// TIA Portal V20 export
// export: Created 2025-12-01T14:57:27.0344131Z, ExportSetting None, DisplayName Totally Integrated Automation Portal, DisplayVersion V20 Update 3, DisplayName TIA Portal Openness, DisplayVersion V20 Update 3, DisplayName TIA Portal Version Control Interface, DisplayVersion V20 Update 3, DisplayName STEP 7 Professional, DisplayVersion V20 Update 3, DisplayName STEP 7 Safety, DisplayVersion V20 Update 2, DisplayName WinCC Basic/Comfort/Advanced, DisplayVersion V20 Update 3, DisplayName WinCC Professional, DisplayVersion V20 Update 3, DisplayName WinCC Unified, DisplayVersion V20 Update 3
FUNCTION "FC608_CambioEstado_Peines" : Void   // FC608, LAD
{ S7_Optimized_Access := 'TRUE' }
// stored: AutoNumber false, SetENOAutomatically false
   VAR_INPUT
      Aplica_Cambio : Bool;
      ID_Quimarox : UInt;
      ID_Peine : UInt;   // Numero_Peine o 999 para ejecutar acción sobre todos los peines
      Acción : UInt;   // 1 Habilitar, 2 Deshabilitar
   END_VAR
   VAR_OUTPUT
      Result : Bool;   // 0 resultado ok, 1 resultado nook
   END_VAR
   VAR_TEMP
      Aux_Contador : UInt;
   END_VAR
BEGIN

NETWORK
TITLE = 0 resultado ok, 1 resultado nook
//======================================================================
// Hasta que no tengamos aplicar cambio, no ejecutamos ninguna acción

      SET;
      AN    #Aplica_Cambio;
      JC    Fin;

//======================================================================
// si la acción es 0, no tenemos que hacer nada

      SET;
      L     #Acción;
      L     0;
      ==I;
      JC    Fin;

//======================================================================
// comprobamos si el ID de quimarox es válido
      SET;
      A(;
      L     #ID_Quimarox;
      L     0;
      <>I;
      );
      A(;
      L     #ID_Quimarox;
      L     "CTE_MaxNumQuimarox";
      <=I;
      );
      JC    rango_quimarox_valido;

//======================================================================
// si el rango no es válido, marcamos result 1 y salimos de la funcióm
      JU    Fin_nok;

//======================================================================
// comprobamos si la acción es sobre un peine o sobre todos
rango_quimarox_valido:NOP   0;

      SET;
      L     #ID_Peine;
      L     999;
      ==I;
      JC    todos_los_peines;

// si la acción no es sobre todos los peines, pasamos a comprobar si el número de peine es válido

      SET;
      A(;
      L     #ID_Peine;
      L     0;
      >I;
      );
      A(;
      L     #ID_Peine;
      L     "DB600_ConfigQuimarox".Quimarox[#ID_Quimarox].datos_config.Numero_vagones;
      <=I;
      );
      JC    rango_peine_valido;
//======================================================================
// si el rango no es válido, marcamos result 1 y salimos de la funcióm

      JU    Fin_nok;

//======================================================================

NETWORK
TITLE = Ejecución de acciones sobre todos los peines
//======================================================================
todos_los_peines:NOP   0;

// inicializamos el contador para movernos por el bucle
      L     1;
      T     #Aux_Contador;

// en función de la acción a ejecutar, vamos a un bucle o a otro
//======================================================================
bucle:L     #Acción;
      JL    LSTX;
      JU    Fin;
      JU    Habilitar_todos;
      JU    Deshabilitar_todos;

LSTX: JU    Fin;
//======================================================================
Habilitar_todos:NOP   0;
      CLR;
      =     "DB601_PeinesQuimarox".Quimarox[#ID_Quimarox].vagon[#Aux_Contador].carrier_no_utilizable;
      JU    Siguiente_Peine;

//======================================================================
Deshabilitar_todos:NOP   0;
      SET;
      =     "DB601_PeinesQuimarox".Quimarox[#ID_Quimarox].vagon[#Aux_Contador].carrier_no_utilizable;
      JU    Siguiente_Peine;
//======================================================================

Siguiente_Peine:NOP   0;
// comprobamos si hemos llegado al final del bucle
      SET;
      L     #Aux_Contador;
      L     "DB600_ConfigQuimarox".Quimarox[#ID_Quimarox].datos_config.Numero_vagones;
      >=I;
      JC    Fin_ok;

// si no hemos acabado, pasamos al siguiente peine

      L     #Aux_Contador;
      L     1;
      +I;
      T     #Aux_Contador;
      JU    bucle;

//======================================================================

NETWORK
TITLE = Ejecución de acciones sobre un peine en concreto
rango_peine_valido:NOP   0;



      L     #Acción;
      JL    LSTXp;
      JU    Fin;
      JU    Habilitar;
      JU    Deshabilitar;

LSTXp:JU    Fin;

//======================================================================
Habilitar:NOP   0;
      CLR;
      =     "DB601_PeinesQuimarox".Quimarox[#ID_Quimarox].vagon[#ID_Peine].carrier_no_utilizable;
      JU    Fin_ok;

//======================================================================
Deshabilitar:NOP   0;
      SET;
      =     "DB601_PeinesQuimarox".Quimarox[#ID_Quimarox].vagon[#ID_Peine].carrier_no_utilizable;
      JU    Fin_ok;
//======================================================================



NETWORK
TITLE = 0 resultado ok, 1 resultado nook
//======================================================================
Fin:  BE;
//======================================================================
Fin_nok:NOP   0;
      SET;
      =     #Result;
      BE;
//======================================================================
Fin_ok:NOP   0;
      CLR;
      =     #Result;
      BE;
//======================================================================
END_FUNCTION
